    |     l2delyunit = struct1[7]
    | 
    |     # FIND THE POINTS ON THE LINES OF THE FIRST TURN PATH
    |     # find locations 8 inches away from  intersect point
    |     # CONST
    |     welddistance1 = 6 # first path first leg (down)
    |     welddistance2 = 4 # first path second leg (under) # inches
    |     welddistance3 = 6 # second path (back away) # inches
    | 
    |     wd1 = welddistance1 * 25.4 / 1000
    |     wd2 = welddistance2 * 25.4 / 1000
    |     wd3 = welddistance3 * 25.4 / 1000
    |     leftwallthickmm = leftwallthick * 25.4 / 1000 # in this step corner right, this is distance from left edge
    |     rightwallthickmm =  rightwallthick * 25.4 / 1000 # in this step corner right, this is distance from right edge
    | 
    |     # first, check if we need a lift column raise
    |     # (we do, because for maximum reach we want to make the lift pedestal be even with the top of the covers)
    |     zpi = pointintersect[2]
    |     if zpi > 0:
    |         liftcolumnzneeded = zpi * 1000.0 # the robot uses coordinates in meters, but the lift column uses coordinates in mm
    |         z = 0
    |     else:
    |         z = zpi
    |     end
    | 
    |     # first, calculate the location of the top of the vertical chamfer (where point2 would be if there weren't any circle motion)
    |     x = pointintersect[0] + l2delxunit * rightwallthickmm
    |     y = pointintersect[1] + l2delyunit * rightwallthickmm
    |     #z = pointintersect[2] # replaced by z of lift column (directly above)
    |     pointtopvcham = p[x, y, z, 0, 0, 0]
    | 
    |     # calculate the rxryrz for the gun when it's at point1
    |     # start with rxryrz = 0,0,0 (gun facing up, preheat facing y+ axis.
    |     # rotate it 180 degrees about x axis. gun facing down, preheat facing y- axis
    |     # rotate it about 45 degrees ccw about z axis. x+ to heading1 is about 135 degrees. so our angle is heading1 - 90 degrees
    |     m1 = get_rotation_matrix_from_description("x", -1, 180 * pi / 180) # rotation 1: 180 degrees forward about x axis
    |     m2 = get_rotation_matrix_from_description("z", 1, heading1 - pi/2) # rotation 2
    |     m3 = multiply_matrix(m2, m1) #we rotate m1 first then m2, so we multiply in backwards order: 2 then 1
    |     rxryrz = convert_matrix_to_axang(m3)
    |     rx = rxryrz[0]
    |     ry = rxryrz[1]
    |     rz = rxryrz[2]
    | 
    |     # next, calculate point1
    |     p1x = x + l1delxunit * wd1
    |     p1y = y + l1delyunit * wd1
    |     point1 = p[p1x, p1y, z, rx, ry, rz]
    | 
    |     # the round over distance is the distance from pointbottomvcham to point2 (which will be the same as distance to p4)
    |     roundoverdistance = 0.05
    |     rod = roundoverdistance * 25.4 / 1000
    |     p2x = x + l1delxunit * rod
    |     p2y = y + l1delyunit * rod
    |     point2 = p[p2x, p2y, z, rx, ry, rz]
    | 
    |     # make point2a, colinear between p1 and p2, which will be the place the welder shuts off during motion
    |     wtod = 0.015 # weldturnoffdistance # meters from pointtopvcham # 10 mm (1.0 seconds)
    |     p2ax = x + l1delxunit * wtod
    |     p2ay = y + l1delyunit * wtod
    |     point2a = p[p2ax, p2ay, z, rx, ry, rz]
    | 
    |     # calculate the rxryrz for facing the down the left side of the box
    |     # rotate about x 90 (forward). then rotate about z ~ 45 (ccw)
    |     m1 = get_rotation_matrix_from_description("x", -1, 90 * pi / 180)
    |     m2 = get_rotation_matrix_from_description("z", 1, heading1 - pi/2)
    |     m3 = multiply_matrix(m2, m1) #we rotate m1 first then m2, so we multiply in backwards order: 2 then 1
    |     rxryrz = convert_matrix_to_axang(m3)
    |     rx = rxryrz[0]
    |     ry = rxryrz[1]
    |     rz = rxryrz[2]
    | 
    |     # calculate point4
    |     point4 = p[x, y, z - rod, rx, ry, rz]
    | 
    |     # calculate point5
    |     point5 = p[x, y, z - wd2, rx, ry, rz]
    | 
    |     # calculate point3
    |     # we know that the angle is exactly 90 degrees
    |     delta = calc_rod_midpoint_90deg(rod)
    |     p3z = z - delta
    |     p3x = x + delta * l1delxunit
    |     p3y = y + delta * l1delyunit
    | 
    |     # calculate rxryrz
    |     m1 = get_rotation_matrix_from_description("x", -1, 135 * pi / 180) # rotation 1: 135 degrees forward about x axis
    |     m2 = get_rotation_matrix_from_description("z", 1, heading1 - pi/2)
    |     m3 = multiply_matrix(m2, m1) #we rotate m1 first then m2, so we multiply in backwards order: 2 then 1
    |     rxryrz = convert_matrix_to_axang(m3)
    |     rx = rxryrz[0]
    |     ry = rxryrz[1]
    |     rz = rxryrz[2]
    |     point3 = p[p3x, p3y, p3z, rx, ry, rz]
    | 
    |     #todo: calculate trail out point
    | 
    |     # calculate back-away (points 201 and 202)
    |     pushtipforward = 0.006 # 6 millimeters forward. the tip needs to clear the capping wall's angled chamfer to not BONK when getting into position
    |     p201x = x + l1delxunit * leftwallthickmm + l2delxunit * pushtipforward
    |     p201y = y + l1delyunit * leftwallthickmm + l2delyunit * pushtipforward
    | 
    |     # calculate rxryrz
    |     # rotate 180 degrees about x. then rotate (90 deg + heading3 degrees) about z ccw
    |     m1 = get_rotation_matrix_from_description("x", -1, 180 * pi / 180)
    |     m2 = get_rotation_matrix_from_description("z", 1, heading3 + pi/2)
    |     m3 = multiply_matrix(m2, m1) #we rotate m1 first then m2, so we multiply in backwards order: 2 then 1
    |     rxryrz = convert_matrix_to_axang(m3)
    |     rx = rxryrz[0]
    |     ry = rxryrz[1]
    |     rz = rxryrz[2]
    |     point201 = p[p201x, p201y, z, rx, ry, rz]
    | 
    |     # calculate point 201's preheat
    |     pushtipforward2 = 0.012 - pushtipforward # 12 mm forward to clear the existing extrudant (but still have the extrudant from this extrusion join the existing). subtract from previous to make it constant even if you change pushtipforward1
    |     preheatdistance = 0.010 # 10 mm . above what it would be pushed down
    |     point201a = p[p201x, p201y, z + preheatdistance, rx, ry, rz]
    |     p201bx = p201x + l2delxunit * pushtipforward2
    |     p201by = p201y + l2delyunit * pushtipforward2
    |     point201b = p[p201bx, p201by, z + preheatdistance, rx, ry, rz]
    |     point201c = p[p201bx, p201by, z, rx, ry, rz]
    | 
    |     # calculate point 202
    |     p202x = p201x + wd3 * l2delxunit
    |     p202y = p201y + wd3 * l2delyunit
    |     point202 = p[p202x, p202y, z, rx, ry, rz]
    | 
    |     struct2 = struct(point1=point1, point2=point2, point3=point3, point4=point4, point5=point5, point201=point201, point202=point202, point201a=point201a, point201b=point201b, point201c=point201c, point2a=point2a)
    |     return struct2
    | end
    | 
    | def calculate_AtS_points_cover_right(struct1, leftwallthick, rightwallthick):
    |     # get the stuff from the struct
    |     pointintersect = struct1[0]
    |     heading1 = struct1[1]
    |     heading2 = struct1[2]
    |     heading3 = struct1[3]
    |     l1delxunit = struct1[4]
    |     l1delyunit = struct1[5]
    |     l2delxunit = struct1[6]
    |     l2delyunit = struct1[7]
    | 
    |     # FIND THE POINTS ON THE LINES OF THE FIRST TURN PATH
    |     # find locations 8 inches away from  intersect point
    |     # CONST
    |     welddistance1 = 6 # first path first leg (down)
    |     welddistance2 = 4 # first path second leg (under) # inches
    |     welddistance3 = 6 # second path (back away) # inches
    | 
    |     wd1 = welddistance1 * 25.4 / 1000
    |     wd2 = welddistance2 * 25.4 / 1000
    |     wd3 = welddistance3 * 25.4 / 1000
    |     leftwallthickmm = leftwallthick * 25.4 / 1000 # in this step corner right, this is distance from left edge
    |     rightwallthickmm =  rightwallthick * 25.4 / 1000 # in this step corner right, this is distance from right edge
    | 
    |     # first, check if we need a lift column raise
    |     # (we do, because for maximum reach we want to make the lift pedestal be even with the top of the covers)
    |     zpi = pointintersect[2]
    |     if zpi > 0:
    |         liftcolumnzneeded = zpi * 1000.0 # the robot uses coordinates in meters, but the lift column uses coordinates in mm
    |         z = 0
    |     else:
    |         z = zpi
    |     end
    | 
    |     # first, calculate the location of the top of the vertical chamfer (where point2 would be if there weren't any circle motion)
    |     x = pointintersect[0] + l1delxunit * leftwallthickmm
    |     y = pointintersect[1] + l1delyunit * leftwallthickmm
    |     #z = pointintersect[2] # replaced by z of lift column (directly above)
    |     pointtopvcham = p[x, y, z, 0, 0, 0]
    | 
    |     # calculate the rxryrz for the gun when it's at point1
    |     # start with rxryrz = 0,0,0 (gun facing up, preheat facing y+ axis.
    |     # rotate it 180 degrees about x axis. gun facing down, preheat facing y- axis
    |     # rotate it about 135 degrees ccw about z axis. x+ to heading3 is about 225 degrees. so our angle is heading3 - 90 degrees
    |     m1 = get_rotation_matrix_from_description("x", -1, 180 * pi / 180) # rotation 1: 180 degrees forward about x axis
    |     m2 = get_rotation_matrix_from_description("z", 1, heading3 - pi/2) # rotation 2
    |     m3 = multiply_matrix(m2, m1) #we rotate m1 first then m2, so we multiply in backwards order: 2 then 1
    |     rxryrz = convert_matrix_to_axang(m3)
    |     rx = rxryrz[0]
    |     ry = rxryrz[1]
    |     rz = rxryrz[2]
    | 
    |     # next, calculate point1
    |     p1x = x + l2delxunit * wd1
    |     p1y = y + l2delyunit * wd1
    |     point1 = p[p1x, p1y, z, rx, ry, rz]
    | 
    |     # the round over distance is the distance from pointbottomvcham to point2 (which will be the same as distance to p4)
    |     roundoverdistance = 0.05
    |     rod = roundoverdistance * 25.4 / 1000
    |     p2x = x + l2delxunit * rod
    |     p2y = y + l2delyunit * rod
    |     point2 = p[p2x, p2y, z, rx, ry, rz]
    | 
    |     # make point2a, colinear between p1 and p2, which will be the place the welder shuts off during motion
    |     wtod = 0.015 # weldturnoffdistance # meters from pointtopvcham # 10 mm (1.0 seconds)
    |     p2ax = x + l2delxunit * wtod
    |     p2ay = y + l2delyunit * wtod
    |     point2a = p[p2ax, p2ay, z, rx, ry, rz]
    | 
    |     # calculate the rxryrz for facing the down the right side of the box
    |     # rotate about x 90 (forward). then rotate about z ~ 135 (ccw)
    |     m1 = get_rotation_matrix_from_description("x", -1, 90 * pi / 180)
    |     m2 = get_rotation_matrix_from_description("z", 1, heading3 - pi/2)
    |     m3 = multiply_matrix(m2, m1) #we rotate m1 first then m2, so we multiply in backwards order: 2 then 1
    |     rxryrz = convert_matrix_to_axang(m3)
    |     rx = rxryrz[0]
    |     ry = rxryrz[1]
    |     rz = rxryrz[2]
    | 
    |     # calculate point4
    |     point4 = p[x, y, z - rod, rx, ry, rz]
    | 
    |     # calculate point5
    |     point5 = p[x, y, z - wd2, rx, ry, rz]
    | 
    |     # calculate point3
    |     # we know that the angle is exactly 90 degrees
    |     delta = calc_rod_midpoint_90deg(rod)
    |     p3z = z - delta
    |     p3x = x + delta * l2delxunit
    |     p3y = y + delta * l2delyunit
    | 
    |     # calculate rxryrz
    |     m1 = get_rotation_matrix_from_description("x", -1, 135 * pi / 180) # rotation 1: 135 degrees forward about x axis
    |     m2 = get_rotation_matrix_from_description("z", 1, heading3 - pi/2)
    |     m3 = multiply_matrix(m2, m1) #we rotate m1 first then m2, so we multiply in backwards order: 2 then 1
    |     rxryrz = convert_matrix_to_axang(m3)
    |     rx = rxryrz[0]
    |     ry = rxryrz[1]
    |     rz = rxryrz[2]
    |     point3 = p[p3x, p3y, p3z, rx, ry, rz]
    | 
    |     #todo: calculate trail out point
    | 
    |     # calculate back-away (points 201 and 202)
    |     pushtipforward = 0.006 # 6 millimeters forward. the tip needs to clear the capping wall's angled chamfer to not BONK when getting into position
    |     p201x = x + l2delxunit * rightwallthickmm + l1delxunit * pushtipforward
    |     p201y = y + l2delyunit * rightwallthickmm + l1delyunit * pushtipforward
    | 
    |     # calculate rxryrz
    |     # rotate 180 degrees about x. then rotate (90 deg + heading1 degrees) about z ccw
    |     m1 = get_rotation_matrix_from_description("x", -1, 180 * pi / 180)
    |     m2 = get_rotation_matrix_from_description("z", 1, heading1 + pi/2)
    |     m3 = multiply_matrix(m2, m1) #we rotate m1 first then m2, so we multiply in backwards order: 2 then 1
    |     rxryrz = convert_matrix_to_axang(m3)
    |     rx = rxryrz[0]
    |     ry = rxryrz[1]
    |     rz = rxryrz[2]
    |     point201 = p[p201x, p201y, z, rx, ry, rz]
    | 
    |     # calculate point 201's preheat
    |     pushtipforward2 = 0.012 - pushtipforward # 12 mm forward to clear the existing extrudant (but still have the extrudant from this extrusion join the existing). subtract from previous to make it constant even if you change pushtipforward1
    |     preheatdistance = 0.010 # 10 mm . above what it would be pushed down
    |     point201a = p[p201x, p201y, z + preheatdistance, rx, ry, rz]
    |     p201bx = p201x + l1delxunit * pushtipforward2
    |     p201by = p201y + l1delyunit * pushtipforward2
    |     point201b = p[p201bx, p201by, z + preheatdistance, rx, ry, rz]
    |     point201c = p[p201bx, p201by, z, rx, ry, rz]
    | 
    |     # calculate point 202
    |     p202x = p201x + wd3 * l1delxunit
    |     p202y = p201y + wd3 * l1delyunit
    |     point202 = p[p202x, p202y, z, rx, ry, rz]
    | 
    |     struct2 = struct(point1=point1, point2=point2, point3=point3, point4=point4, point5=point5, point201=point201, point202=point202, point201a=point201a, point201b=point201b, point201c=point201c, point2a=point2a)
    |     return struct2
    | end
    | 
    | def main_calculate_cover_straight(p11, p12, p21, p22, sidewallthick, leftpoint, rightpoint):
    |     struct1 = analyze_touchpoints_only_cover_straight(p11, p12, p21, p22, leftpoint)
    |     struct2 = calculate_straight_points_cover(struct1, sidewallthick, leftpoint, rightpoint)
    |     #struct2 = calculate_DOtA_points_left_extended(struct1, list1, chamferover, chamferup, tcp_pose_top)
    |     #struct3 = check_validity_left(struct1, struct2)
    |     return struct2
    | 
    | end
    | 
    | # calculates the line of intersection of the sidewall plane (assumed vertical) and the cover plane (assumed perpendicular to sidewall plane)
    | # returns a struct containing point0 (point on the intersection line, same y as leftpoint) and 3 components of the unit vector left to right and 2 components of the other direction in 2d
    | def analyze_touchpoints_only_cover_straight(p11, p12, p21, p22, leftpoint):
    |     # calculate slope of sidewall in x-y plane
    |     # get the raw points from the first line
    |     l1p1x=p11[0]
    |     l1p1y=p11[1]
    |     l1p2x=p12[0]
    |     l1p2y=p12[1]
    | 
    |     # equate the first line in 2d space
    |     ml1 = (l1p2y-l1p1y) / (l1p2x-l1p1x)
    | 
    |     # b = y - mx
    |     bl1 = l1p1y - ml1 * l1p1x
    | 
    |     # calculate the cover plane
    |     # if two planes are perpendicular, then their normal vectors must be perpendicular.
    |     # the first planes normal vector is n1, which is taken from the equation of the plane ax + by + cz = d -> <a, b, c>
    |     # the second plane's normal vector is perpendicular to all vectors contained in the plane
    |     # p21 to p22 is a vector v contained within plane 2.
    |     # n2 is normal to both n1 AND v. to achieve a vector that is normal to both, take the cross product
    | 
    |     # plane 1 (y = mx + b) -> (b = -mx +1y +0z)
    |     n1 = [-1 * ml1, 1, 0]
    | 
    |     # v=P2−P1=(x2−x1,y2−y1,z2−z1)
    |     v = [p21[0]-p22[0], p21[1]-p22[1], p21[2]-p22[2]]
    | 
    |     #v n2 = cross product of n1 and v
    |     n2x = n1[1]*v[2] - n1[2]*v[1]
    |     n2y = n1[2]*v[0] - n1[0]*v[2]
    |     n2z = n1[0]*v[1] - n1[1]*v[0]
    |     n2 = [n2x, n2y, n2z]
    | 
    |     # find the d of the second plane
    |     # n2x * x + n2y * y + n2z * z = d0
    |     d = n2x * p21[0] + n2y * p21[1] + n2z * p21[2]
    | 
    |     # find the intersection line of the two planes
    |     # find the direction vector of that line by taking the cross product of the normal vector of those two planes
    |     v3x = n1[1]*n2[2] - n1[2]*n2[1]
    |     v3y = n1[2]*n2[0] - n1[0]*n2[2]
    |     v3z = n1[0]*n2[1] - n1[1]*n2[0]
    |     v3 = [v3x, v3y, v3z]
    | 
    |     # normalize the vector so the magnitude is 1
    |     magnitude2 = v3x * v3x + v3y * v3y + v3z * v3z
    |     magnitude = sqrt(magnitude2)
    |     v3xunit = v3x/magnitude
    |     v3yunit = v3y/magnitude
    |     v3zunit = v3z/magnitude
    | 
    |     # make sure it is going the right way (from left to right). make sure the v3yunit is positive
    |     if v3yunit < 0:
    |         v3xunit = v3xunit * -1
    |         v3yunit = v3yunit * -1
    |         v3zunit = v3zunit * -1
    |     end
    | 
    |     # next we have to find a point on the line by setting one of the dimensions and solving the system of equations
    |     # i will pick the y value of the left teach point
    |     y = leftpoint[1]
    |     # plane 1: -ml1 * x + 1 * y + 0 * z = bl1
    |     # -ml1 * x = bl1 - y
    |     x = (bl1 - y)/ (-1 * ml1)
    |     # plane 2: d = n2x * x + n2y * y + n2z * z
    |     # (d - n2x * x - n2y * y) = n2z * z
    |     z = (d - n2x * x - n2y * y) / n2z
    | 
    |     # make point0 into a pose
    |     point0 = p[x, y, z, 0, 0, 0]
    | 
    |     # find heading of main line
    |     heading1 = convert_uv_to_heading(v3xunit, v3yunit)
    | 
    |     # make a unit vector perpendicular to this one in the xy plane pointing x -. will be used to move over the chamfer distance
    |     ml2 = -1 / ml1
    |     # y = ml2 * x + unknownB
    |     # vector = [1, ml2]
    |     mag2 = 1 + ml2 * ml2
    |     mag = sqrt(mag2)
    |     v4xunit = 1 / mag
    |     v4yunit = ml2 / mag
    |     # switch is to the x direction is negative
    |     v4xunit = -1 * v4xunit
    |     v4yunit = -1 * v4yunit
    | 
    |     ret = struct(point0=point0, v3xunit=v3xunit, v3yunit=v3yunit, v3zunit=v3zunit, heading1=heading1, v4xunit=v4xunit, v4yunit=v4yunit)
    |     return ret
    | end
    | 
    | def calculate_straight_points_cover(struct1, sidewallthick, leftpointteach, rightpointteach):
    |     # get the stuff
    |     point0 = struct1[0]
    |     p0x = point0[0]
    |     p0y = point0[1]
    |     p0z = point0[2]
    |     v3xunit = struct1[1]
    |     v3yunit = struct1[2]
    |     v3zunit = struct1[3]
    |     heading1 = struct1[4]
    |     v4xunit = struct1[5]
    |     v4yunit = struct1[6]
    |     sidewallthick = sidewallthick
    |     lpy = leftpointteach[1]
    |     rpy = rightpointteach[1]
    | 
    |     # first, check if we need a lift column raise
    |     # (we do, because for maximum reach we want to make the lift pedestal be even with the top of the covers)
    |     zpi = p0z
    |     if zpi > 0:
    |         liftcolumnzneeded = zpi * 1000.0 # the robot uses coordinates in meters, but the lift column uses coordinates in mm
    |         coverz = 0
    |     else:
    |         coverz = zpi
    |     end
    | 
    |     # calculate pointtopvcham
    |     chamferover = sidewallthick * 25.4 / 1000.0
    |     tiltraise = 0.006 # 6 mm raise needed for the tip to clear the plane during tiltback
    |     x = p0x + v4xunit * chamferover
    |     y = p0y + v4yunit * chamferover
    |     z = coverz + tiltraise
    | 
    |     # calculate rxryrz for tilted back
    |     # 3 rotations to make this happen.
    |     # start point is straight up with the preheat pointed in the +y direction.
    |     # first rotation is 180 degrees about x direction. gun is now pointing straight down with preheat facing -y direction
    |     m1 = get_rotation_matrix_from_description("x", 1, 180 * pi / 180)
    |     # second rotation is a 10 degree turn about the x axis (negative direction)
    |     m2 = get_rotation_matrix_from_description("x", -1, 10 * pi / 180)
    |     # third rotation is about 180 degrees about the z axis. starting from the -y axis, go until you get to heading1. that will equal heading1 plus 90 degrees
    |     m3 = get_rotation_matrix_from_description("z", 1, pi/2 + heading1)
    |     # combine them by multiplying m3 * m2 * m1
    |     # matrix multiplication is not commutative but it IS associative, so you can do this whichever order
    |     m4 = multiply_matrix(m2, m1)
    |     m5 = multiply_matrix(m3, m4)
    |     rxryrzt = convert_matrix_to_axang(m5)
    |     rxt = rxryrzt[0]
    |     ryt = rxryrzt[1]
    |     rzt = rxryrzt[2]
    |     pointtopvcham = p[x, y, z, rxt, ryt, rzt]
    | 
    |     # calculate point1 (preheat)
    |     dist = -1 * 25.4 / 1000.0 # move back 1 inch from
    |     p1x = x + dist * v3xunit
    |     p1y = y + dist * v3yunit
    |     p1z = z + dist * v3zunit
    |     point1 = p[p1x, p1y, p1z, rxt, ryt, rzt]
    | 
    |     # calculate point2 (start of flatten)
    |     dist = 0.5 * 25.4 / 1000.0  # half an inch past the top of v chamfer
    |     p2x = x + dist * v3xunit
    |     p2y = y + dist * v3yunit
    |     p2z = z + dist * v3zunit
    |     point2 = p[p2x, p2y, p2z, rxt, ryt, rzt]
    | 
    |     # calculate rxryrz for nontilted
    |     # first rotation is 180 degrees about x direction. gun is now pointing straight down with preheat facing -y direction
    |     m1 = get_rotation_matrix_from_description("x", 1, 180 * pi / 180)
    |     # third rotation is about 180 degrees about the z axis. starting from the -y axis, go until you get to heading1. that will equal heading1 plus 90 degrees
    |     m3 = get_rotation_matrix_from_description("z", 1, pi/2 + heading1)
    |     m5 = multiply_matrix(m3, m1)
    |     rxryrz = convert_matrix_to_axang(m5)
    |     rx = rxryrz[0]
    |     ry = rxryrz[1]
    |     rz = rxryrz[2]
    | 
    |     # calculate point3 (end of flatten)
    |     dist = 1.5 * 25.4 / 1000.0  # 1.5 inches past top of v chamfer
    |     p3x = x + dist * v3xunit
    |     p3y = y + dist * v3yunit
    |     p3z = coverz + dist * v3zunit
    |     point3 = p[p3x, p3y, p3z, rx, ry, rz]
    | 
    |     # calculate distance between leftpoint and rightpoint
    |     # we have the y distance. we need to find the total distance.
    |     # the unit vector (v3) should have a magnitude of 1. that's what analyze_touchpoints_only_cover_straight() calculated.
    |     # so the total distance is y distance * 1 / v3yunit
    |     ydist = rpy - lpy
    |     totdist = ydist / v3yunit
    | 
    |     # calculate pointtopvcham2
    |     x2 = x + v3xunit * totdist
    |     y2 = y + v3yunit * totdist
    |     z2 = z + v3zunit * totdist
    | 
    |     # calculate point4 (start of unflatten)
    |     dist = -1.5 * 25.4 / 1000.0
    |     p4x = x2 + v3xunit * dist
    |     p4y = y2 + v3yunit * dist
    |     p4z = z2 + v3zunit * dist - tiltraise
    |     point4 = p[p4x, p4y, p4z, rx, ry, rz]
    | 
    |     # calculate point5 (end of unflatten)
    |     dist = -0.5 * 25.4 / 1000.0
    |     p5x = x2 + v3xunit * dist
    |     p5y = y2 + v3yunit * dist
    |     p5z = z2 + v3zunit * dist
    |     point5 = p[p5x, p5y, p5z, rxt, ryt, rzt]
    | 
    |     # calculate point6 (end of smear)
    |     dist = 2 * 25.4 / 1000.0
    |     p6x = x2 + v3xunit * dist
    |     p6y = y2 + v3yunit * dist
    |     p6z = z2 + v3zunit * dist
    |     point6 = p[p6x, p6y, p6z, rxt, ryt, rzt]
    | 
    | 
    |     # return struct
    |     ret = struct(pointtopvcham=pointtopvcham, point1=point1, point2=point2, point3=point3, point4=point4, point5=point5, point6=point6)
    |     return ret
    | 
    | 
    | end
  path_pre := get_straight_homing_pathpoints_floor(tcp_pose_left,tcp_pose_right)
  ph1 := path_pre[0]
  ph2 := path_pre[1]
  ph3 := path_pre[2]
  ph4 := path_pre[3]
  ph4a := p[ph4[0]+0.1,ph4[1],ph4[2],ph4[3],ph4[4],ph4[5]]
  MoveL speed 250 mm/s, acceleration 1200 mm/s^2 (useActiveTCP=true optimoveEnabled=false optiMoveSpeed=0.3 optiMoveAcceleration=0.09) feature=Base
    MoveDirectionNode (selectedDirection=XPlus)
      Until DISTANCE (allowActions=false deceleration=3 distanceNodeType=STOP) Distance=0.1; motionParameters(blendRadius=0)
  MoveJ speed 60 deg/s, acceleration 80 deg/s^2 (useActiveTCP=true optimoveEnabled=false optiMoveSpeed=0.3 optiMoveAcceleration=0.09) feature=Base
    SuppressedNode
      Waypoint Waypoint_11: TCP in base x=-589.354 y=-454.462 z=658.693 mm, rx=1.8664 ry=-1.8664 rz=-0.5984 rad; joints [32.16, -93.601, 92.579, 59.83, 108.044, 27.179] deg; TCP offset x=-1.032 y=-18.062 z=285.234 mm, rx=0 ry=0 rz=0 rad
    Waypoint Waypoint_1: TCP in base x=-589.354 y=-224.033 z=519.728 mm, rx=1.0077 ry=-1.3585 rz=-1.2216 rad; joints [24.032, -118.039, 143.045, -26.295, 122.645, 7.654] deg
  MoveL speed 250 mm/s, acceleration 200 mm/s^2 (useActiveTCP=true optimoveEnabled=false optiMoveSpeed=0.3 optiMoveAcceleration=0.09) feature=Base
    Waypoint Variable (Variable): variable=ph1
  MoveL speed 20 mm/s, acceleration 100 mm/s^2 (useActiveTCP=true optimoveEnabled=false optiMoveSpeed=0.3 optiMoveAcceleration=0.09) feature=Base
    MoveDirectionNode (selectedDirection=XMinus)
      Until TOOL_CONTACT_DETECTION (allowActions=false retraction=0 decelerationAcceleration=3 decelerationAngularAcceleration=34.906585)
  p11 := get_actual_tcp_pose()
  MoveJ speed 60 deg/s, acceleration 80 deg/s^2 (useActiveTCP=true optimoveEnabled=false optiMoveSpeed=0.3 optiMoveAcceleration=0.09) feature=Base
    Waypoint Variable (Variable): variable=ph1
    Waypoint Variable (Variable): variable=ph2
  MoveL speed 20 mm/s, acceleration 100 mm/s^2 (useActiveTCP=true optimoveEnabled=false optiMoveSpeed=0.3 optiMoveAcceleration=0.09) feature=Base
    MoveDirectionNode (selectedDirection=XMinus)
      Until TOOL_CONTACT_DETECTION (allowActions=false retraction=0 decelerationAcceleration=3 decelerationAngularAcceleration=34.906585)
  SuppressedNode
    p13 := get_actual_tcp_pose()
  SuppressedNode
    MoveJ speed 60 deg/s, acceleration 80 deg/s^2 (useActiveTCP=true optimoveEnabled=false optiMoveSpeed=0.3 optiMoveAcceleration=0.09) feature=Base
      Waypoint Variable (Variable): variable(name=ph2up)
      Waypoint Variable (Variable): variable=ph3
  SuppressedNode
    MoveL speed 20 mm/s, acceleration 100 mm/s^2 (useActiveTCP=true optimoveEnabled=false optiMoveSpeed=0.3 optiMoveAcceleration=0.09) feature=Base
      MoveDirectionNode expression=[-1,-1.0,0.0]
        Until TOOL_CONTACT_DETECTION (allowActions=false retraction=0 decelerationAcceleration=3 decelerationAngularAcceleration=34.906585)
  p12 := get_actual_tcp_pose()
  MoveJ speed 60 deg/s, acceleration 80 deg/s^2 (useActiveTCP=true optimoveEnabled=false optiMoveSpeed=0.3 optiMoveAcceleration=0.09) feature=Base
    Waypoint Variable (Variable): variable=ph2
  MoveJ speed 60 deg/s, acceleration 80 deg/s^2 (useActiveTCP=true optimoveEnabled=false optiMoveSpeed=0.3 optiMoveAcceleration=0.09) feature=Base
    Waypoint Variable (Variable): variable=ph1
  MoveJ speed 60 deg/s, acceleration 80 deg/s^2 (useActiveTCP=true optimoveEnabled=false optiMoveSpeed=0.3 optiMoveAcceleration=0.09) feature=Base
    SuppressedNode
      Waypoint Waypoint_11: TCP in base x=-589.354 y=-454.462 z=658.693 mm, rx=1.8664 ry=-1.8664 rz=-0.5984 rad; joints [32.16, -93.601, 92.579, 59.83, 108.044, 27.179] deg
    Waypoint Waypoint_3: TCP in base x=-589.354 y=-224.033 z=519.728 mm, rx=1.0077 ry=-1.3585 rz=-1.2216 rad; joints [24.032, -118.039, 143.045, -26.295, 122.645, 7.654] deg
    SuppressedNode
      Waypoint Waypoint_3: TCP in base x=-1381.315 y=-113.246 z=483.261 mm, rx=0.347 ry=3.1015 rz=-0.0385 rad; joints [-4.848, -55.573, 57.279, 269.477, -88.568, -82.096] deg
    SuppressedNode
      Waypoint Waypoint_9: TCP in base x=-594.234 y=-418.092 z=645.151 mm, rx=0.1258 ry=-0.6986 rz=-0.4993 rad; joints [32.009, -82.779, 153.256, -126.399, 112.73, 35.158] deg
    SuppressedNode
      Waypoint Waypoint_6: TCP in base x=-563.856 y=-113.246 z=483.261 mm, rx=0.347 ry=3.1015 rz=-0.0385 rad; joints [-12.028, -113.359, 121.362, 263.351, -88.693, -89.284] deg
    SuppressedNode
      Waypoint Waypoint_15: TCP in base x=-841.932 y=-252.174 z=466.323 mm, rx=-0.1894 ry=-0.3294 rz=0.1013 rad; joints [8.59, -43.671, 136.758, -165.147, 102.406, 89.233] deg
    SuppressedNode
      Waypoint Waypoint_8: TCP in base x=-869.439 y=-409.581 z=418.615 mm, rx=0 ry=-0.0001 rz=0 rad; joints [12.101, -33.012, 119.104, -176.134, 89.938, 77.897] deg
    SuppressedNode
      Waypoint Waypoint_12: TCP in base x=-1028.087 y=-409.581 z=-52.555 mm, rx=0 ry=-0.0001 rz=0.7467 rad; joints [10.416, 0.258, 83.964, -174.263, 89.923, 122.381] deg
    SuppressedNode
      Waypoint Waypoint_13: TCP in base x=-867.034 y=98.846 z=-52.555 mm, rx=0 ry=-0.0001 rz=0.7467 rad; joints [-20.439, 1.166, 101.357, -192.565, 89.913, 153.243] deg
    Waypoint Waypoint_17: TCP in base x=-574.647 y=213.551 z=642.998 mm, rx=-0.2366 ry=-0.9664 rz=-0.9158 rad; joints [-39.25, -121.471, 159.271, -73.052, 92.515, 73.526] deg
    Waypoint Waypoint_16: TCP in base x=-343.952 y=632.142 z=615.175 mm, rx=-0.0259 ry=-0.0088 rz=-0.5675 rad; joints [-78.579, -51.22, 142.034, -179.331, 90.185, 136.06] deg
  SuppressedNode
    MoveJ speed 60 deg/s, acceleration 80 deg/s^2 (useActiveTCP=true optimoveEnabled=false optiMoveSpeed=0.3 optiMoveAcceleration=0.09) feature=Base
      Waypoint Waypoint_4: TCP in base x=-658.265 y=299.53 z=30.91 mm, rx=0.4268 ry=-1.6215 rz=0.4371 rad; joints [-77.363, -55.591, 142.792, -102.186, -19.322, 105.94] deg; TCP offset x=0 y=0 z=246 mm, rx=0 ry=0 rz=0 rad
      Waypoint Waypoint_5: TCP in base x=-448.863 y=524.6 z=-175.967 mm, rx=2.4733 ry=-1.8744 rz=0.2053 rad; joints [-65.056, -57.525, 139.86, -164.756, -91.924, 99.291] deg
      SuppressedNode
        Waypoint Waypoint_5: TCP in base x=-542.919 y=212.782 z=86.75 mm, rx=-0.746 ry=-1.5701 rz=-0.8083 rad; joints [-15.32, -63.738, 160.053, -88.648, -229.235, 89.501] deg
      Waypoint Waypoint_10: TCP in base x=-559.13 y=259.234 z=102.446 mm, rx=-0.8226 ry=-1.4861 rz=-0.8815 rad; joints [-31.871, -61.56, 166.811, -101.777, -239.831, 87.599] deg; TCP offset x=-1.157 y=-95.604 z=257.595 mm, rx=0 ry=0 rz=0 rad
  MoveL speed 250 mm/s, acceleration 1200 mm/s^2 (useActiveTCP=true optimoveEnabled=false optiMoveSpeed=0.3 optiMoveAcceleration=0.09) feature=Base
    Waypoint Variable (Variable): variable=ph4a
    Waypoint Variable (Variable): variable=ph3
  MoveL speed 20 mm/s, acceleration 100 mm/s^2 (useActiveTCP=true optimoveEnabled=false optiMoveSpeed=0.3 optiMoveAcceleration=0.09) feature=Base
    MoveDirectionNode (selectedDirection=ZPlus)
      Until TOOL_CONTACT_DETECTION (allowActions=false retraction=0 decelerationAcceleration=3 decelerationAngularAcceleration=34.906585)
  p21 := get_actual_tcp_pose()
  MoveL speed 250 mm/s, acceleration 1200 mm/s^2 (useActiveTCP=true optimoveEnabled=false optiMoveSpeed=0.3 optiMoveAcceleration=0.09) feature=Base
    Waypoint Variable (Variable): variable=ph3
  MoveJ speed 60 deg/s, acceleration 80 deg/s^2 (useActiveTCP=true optimoveEnabled=false optiMoveSpeed=0.3 optiMoveAcceleration=0.09) feature=Base
    Waypoint Variable (Variable): variable=ph4
  MoveL speed 20 mm/s, acceleration 100 mm/s^2 (useActiveTCP=true optimoveEnabled=false optiMoveSpeed=0.3 optiMoveAcceleration=0.09) feature=Base
    MoveDirectionNode (selectedDirection=ZPlus)
      Until TOOL_CONTACT_DETECTION (allowActions=false retraction=0 decelerationAcceleration=3 decelerationAngularAcceleration=34.906585)
  p22 := get_actual_tcp_pose()
  MoveL speed 250 mm/s, acceleration 1200 mm/s^2 (useActiveTCP=true optimoveEnabled=false optiMoveSpeed=0.3 optiMoveAcceleration=0.09) feature=Base
    Waypoint Variable (Variable): variable=ph4
    Waypoint Variable (Variable): variable=ph4a
    MoveJ speed 60 deg/s, acceleration 80 deg/s^2 (useActiveTCP=true optimoveEnabled=false optiMoveSpeed=0.3 optiMoveAcceleration=0.09) feature=Base
      Waypoint Waypoint_16: TCP in base x=-343.952 y=632.142 z=615.175 mm, rx=-0.0259 ry=-0.0088 rz=-0.5675 rad; joints [-78.579, -51.22, 142.034, -179.331, 90.185, 136.06] deg; TCP offset x=-1.032 y=-18.062 z=285.234 mm, rx=0 ry=0 rz=0 rad
  SuppressedNode
    MoveJ speed 60 deg/s, acceleration 80 deg/s^2 (useActiveTCP=true optimoveEnabled=false optiMoveSpeed=0.3 optiMoveAcceleration=0.09) feature=Base
      Waypoint Variable (Variable): variable(name=ph7)
      Waypoint Variable (Variable): variable(name=ph6)
      Waypoint Waypoint_14: TCP in base x=-343.952 y=632.142 z=615.175 mm, rx=-0.0259 ry=-0.0088 rz=-0.5675 rad; joints [-77.363, -55.591, 142.791, -175.721, 90.298, 134.942] deg; TCP offset x=0 y=0 z=246 mm, rx=0 ry=0 rz=0 rad
      Waypoint Waypoint_4: TCP in base x=-658.265 y=299.53 z=30.91 mm, rx=0.4268 ry=-1.6215 rz=0.4371 rad; joints [-77.363, -55.591, 142.792, -102.186, -19.322, 105.94] deg
      Waypoint Waypoint_41: TCP in base x=392.128 y=533.269 z=644.149 mm, rx=0.0578 ry=2.126 rz=2.134 rad; joints [-198.126, -117.852, 133.303, -13.01, -11.421, -6.036] deg; TCP offset x=0 y=-4 z=284 mm, rx=0 ry=0 rz=0 rad
      'above waypoint is home'
  SafeHome (positionOptionType=SPEED_AND_ACCELERATION speed=1.047198 acceleration=1.396263 nextMotionTime=2)
